// Mitsubishi GX Works2 project: PLCֹֹֹ_GROUP_31.docx   PLC: FX3G

// global labels: Global1
VAR_GLOBAL
  SW_DAY_START AT X007 : BOOL;
  RESET_ALL AT M10 : BOOL;
  DAY_ACTIVE AT M0 : BOOL;
  SW_EMERGENCY AT X005 : BOOL;
  LAMP_WORK_DAY AT Y007 : BOOL;
  INIT_RASPBERRY AT D1100 : REAL;
  INIT_LEMON AT D1110 : REAL;
  INIT_STABILIZER AT D1120 : REAL;
  INIT_GUMMIES AT D1130 : REAL;
  STOCK_RASPBERRY AT D1200 : REAL;
  STOCK_LEMON AT D1210 : REAL;
  STOCK_STABILIZER AT D1220 : REAL;
  STOCK_GUMMIES AT D1230 : REAL;
  SW_START_PROCESS AT X001 : BOOL;
  PHASE_PREPARE AT M2 : BOOL;
  PHASE_COOL AT M3 : BOOL;
  PHASE_MIX AT M4 : BOOL;
  ANALOG_IN1 AT D8280 : INT;
END_VAR
VAR_GLOBAL CONSTANT
  Constant_5 : REAL := 5;
END_VAR
VAR_GLOBAL
  TYPE_REGULAR AT M1 : BOOL;
END_VAR
VAR_GLOBAL CONSTANT
  Constant_6 : REAL := 6;
END_VAR
VAR_GLOBAL
  PROCESS_TRIGGER AT M6 : BOOL;
END_VAR
VAR_GLOBAL CONSTANT
  Constant_280 : REAL := 280;
  Constant_455 : REAL := 455;
  Constant_105 : REAL := 105;
  Constant_28 : REAL := 28;
  Constant_385 : REAL := 385;
  Constant_665 : REAL := 665;
  Constant_210 : REAL := 210;
  Constant_70 : REAL := 70;
END_VAR
VAR_GLOBAL
  NEEDED_RASPBERRY AT D1400 : REAL;
  NEEDED_LEMON AT D1410 : REAL;
  NEEDED_STABILIZER AT D1420 : REAL;
  NEEDED_GUMMIES AT D1430 : REAL;
  STOCK_OK AT M5 : BOOL;
  LAMP_PREPARE AT Y000 : BOOL;
  TIMER_PREPARE AT TC0 : BOOL;
  Const_5_sec AT K50 : INT;
  SW_COOL AT X002 : BOOL;
  PREP_RASPBERRY AT D1500 : REAL;
  PREP_LEMON AT D1510 : REAL;
  PREP_STABILIZER AT D1520 : REAL;
  PREP_GUMMIES AT D1530 : REAL;
END_VAR
VAR_GLOBAL CONSTANT
  Constant_35 : REAL := 35;
  Constant_420 : REAL := 420;
END_VAR
VAR_GLOBAL
  NEEDED_RASP_FOR_RASP AT D1800 : REAL;
  NEEDED_LEMON_FOR_RASP AT D1810 : REAL;
  NEEDED_STAB_FOR_RASP AT D1820 : REAL;
  NEEDED_LEMON_FOR_LEMON AT D1900 : REAL;
  NEEDED_STAB_FOR_LEMON AT D1910 : REAL;
END_VAR
VAR_GLOBAL CONSTANT
  Constant_560 : REAL := 560;
  Constant_140 : REAL := 140;
END_VAR
VAR_GLOBAL
  GELATO_RASPBERRY AT D1500 : REAL;
  GELATO_LEMON AT D1510 : REAL;
  COOL_GELATO_RASPBERRY AT D1600 : REAL;
END_VAR
VAR_GLOBAL CONSTANT
  Constant_0 : REAL;
END_VAR
VAR_GLOBAL
  TIMER_COOL AT TC1 : BOOL;
  Const_8_sec AT K80 : INT;
  LAMP_COOL AT Y002 : BOOL;
  TEMP_SENSOR AT X003 : BOOL;
  MIX_TOTAL AT D1700 : REAL;
  FLASH_DIFFERENCES AT M7 : BOOL;
  TIMER_MIX_3 AT TC2 : BOOL;
  Const_3_sec AT K30 : INT;
  LAMP_MIX_A AT Y005 : BOOL;
  Const_05_sec AT K5 : INT;
  TIMER_MIX_05 AT TC2 : BOOL;
  TIMER_MIX_050 AT TC3 : BOOL;
  LAMP_MIX_B AT Y006 : BOOL;
  TIMER_MIX AT TC4 : BOOL;
  STORAGE_COUNT AT D1300 : REAL;
END_VAR
VAR_GLOBAL CONSTANT
  Constant_1 : REAL := 1;
  Constant_10 : REAL := 10;
END_VAR
VAR_GLOBAL
  COOL_GELATO_LEMON AT D1610 : REAL;
  MANUAL_STOP_REQ AT M20 : BOOL;
  STOCK_STOP_REQ AT M21 : BOOL;
  MIX_TIMER_EN AT M8 : BOOL;
  TIMER_MIX_REGULAR AT TC4 : BOOL;
  TIMER_MIX_PINUK AT TC5 : BOOL;
  TS_2 AT TS2 : BOOL;
  TS_3 AT TS3 : BOOL;
  TS_5 AT TS5 : BOOL;
  TS_4 AT TS4 : BOOL;
  TIMER_MIX_REGUL AT TC4 : BOOL;
  TIMER_MIX_05_REGULAR AT TC2 : BOOL;
  TIMER_MIX_050_REGULAR AT TC3 : BOOL;
  TIMER_MIX_05_SPECIAL AT TC6 : BOOL;
  TIMER_MIX_050_SPECIAL AT TC7 : BOOL;
  Const_1_sec AT K10 : INT;
  TIMER_MIX_05_2 AT TC2 : BOOL;
  TIMER_MIX_05_3 AT TC3 : BOOL;
  INPUT AT D2000 : REAL;
END_VAR
VAR_GLOBAL CONSTANT
  Constant_400 : REAL := 400;
  WORD_0 : DINT;
END_VAR
VAR_GLOBAL
  ANALOG_OUT AT D8282 : DINT;
  UPDATE AT M8 : BOOL;
  STORAGE_OUT AT D1310 : REAL;
END_VAR
VAR_GLOBAL CONSTANT
  Constant_10_WORD : DINT := 10;
  Constant_40 : REAL := 40;
  Constant_5_5 : REAL := 5.5;
END_VAR

// task Task_01 (event TRUE, interval 0, priority 31): POU_01

PROGRAM POU_01
(* structured ladder/FBD written out as ST: instructions are called as NAME(EN, inputs, outputs); _pN, _eN, _tN stand for wires *)
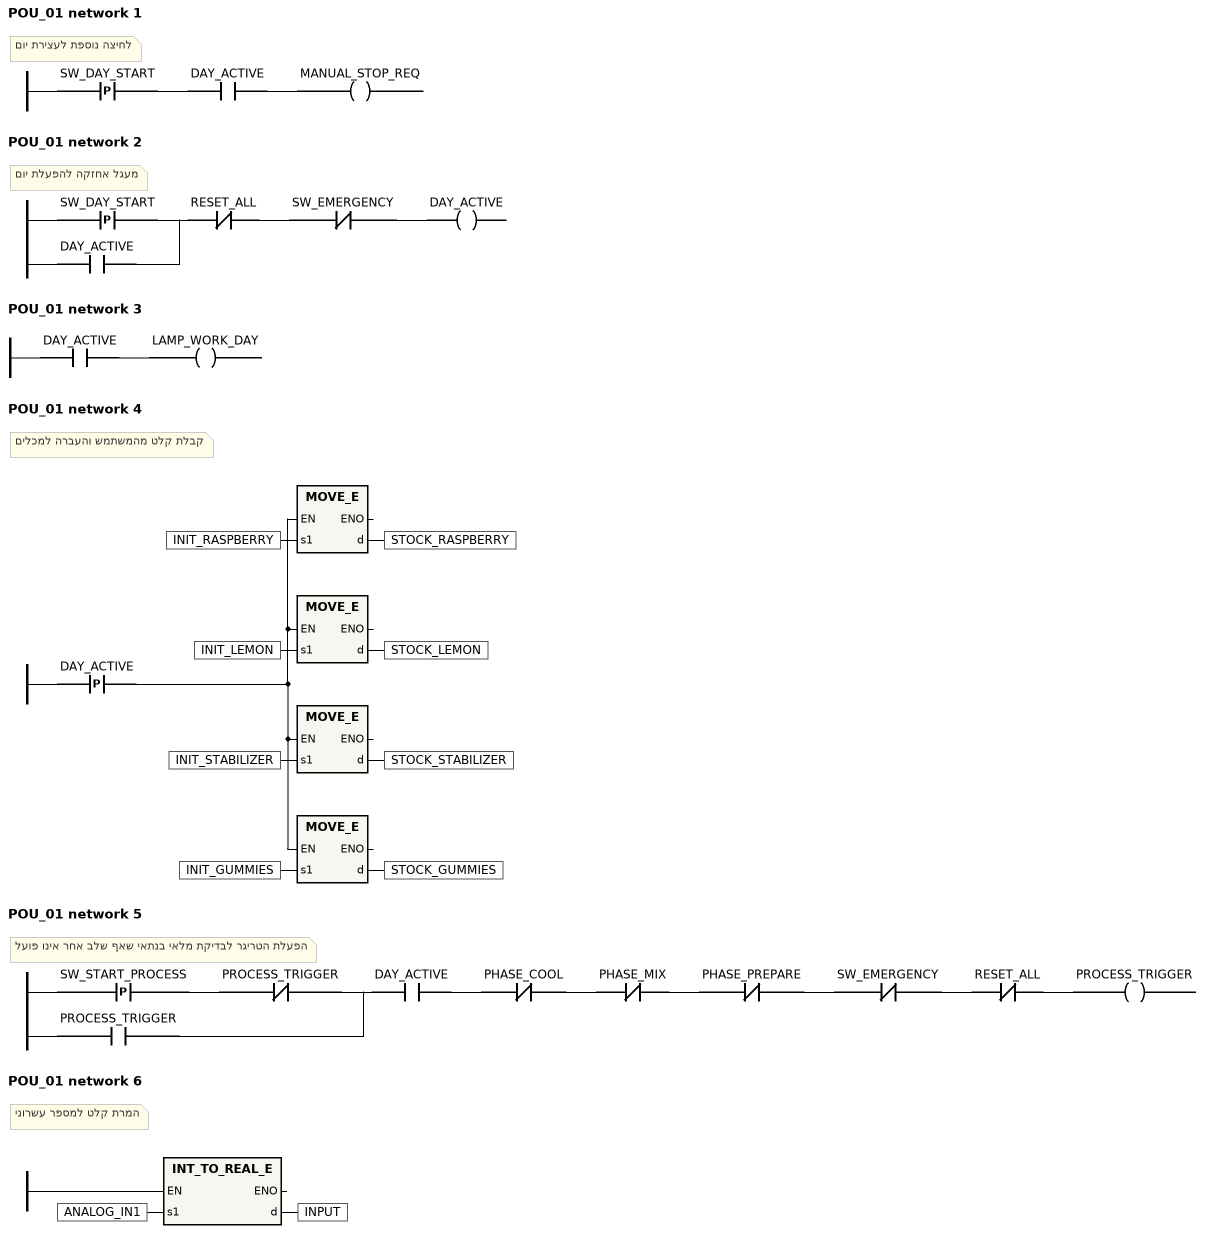
(* network 1 *)
(* לחיצה נוספת לעצירת יום *)
MANUAL_STOP_REQ := LDP(TRUE, SW_DAY_START) AND DAY_ACTIVE;
(* network 2 *)
(* מעגל אחזקה להפעלת יום *)
DAY_ACTIVE := ((LDP(TRUE, SW_DAY_START) OR DAY_ACTIVE) AND NOT RESET_ALL) AND NOT SW_EMERGENCY;
(* network 3 *)
LAMP_WORK_DAY := DAY_ACTIVE;
(* network 4 *)
(* קבלת קלט מהמשתמש והעברה למכלים *)
_p1 := LDP(TRUE, DAY_ACTIVE);
MOVE_E(_p1, INIT_RASPBERRY, STOCK_RASPBERRY);
MOVE_E(_p1, INIT_LEMON, STOCK_LEMON);
MOVE_E(_p1, INIT_STABILIZER, STOCK_STABILIZER);
MOVE_E(_p1, INIT_GUMMIES, STOCK_GUMMIES);
(* network 5 *)
(* הפעלת הטריגר לבדיקת מלאי בנתאי שאף שלב אחר אינו פועל *)
PROCESS_TRIGGER := (((((((LDP(TRUE, SW_START_PROCESS) AND NOT PROCESS_TRIGGER) OR PROCESS_TRIGGER) AND DAY_ACTIVE) AND NOT PHASE_COOL) AND NOT PHASE_MIX) AND NOT PHASE_PREPARE) AND NOT SW_EMERGENCY) AND NOT RESET_ALL;
(* network 6 *)
(* המרת קלט למספר עשרוני *)
INT_TO_REAL_E(TRUE, ANALOG_IN1, INPUT);
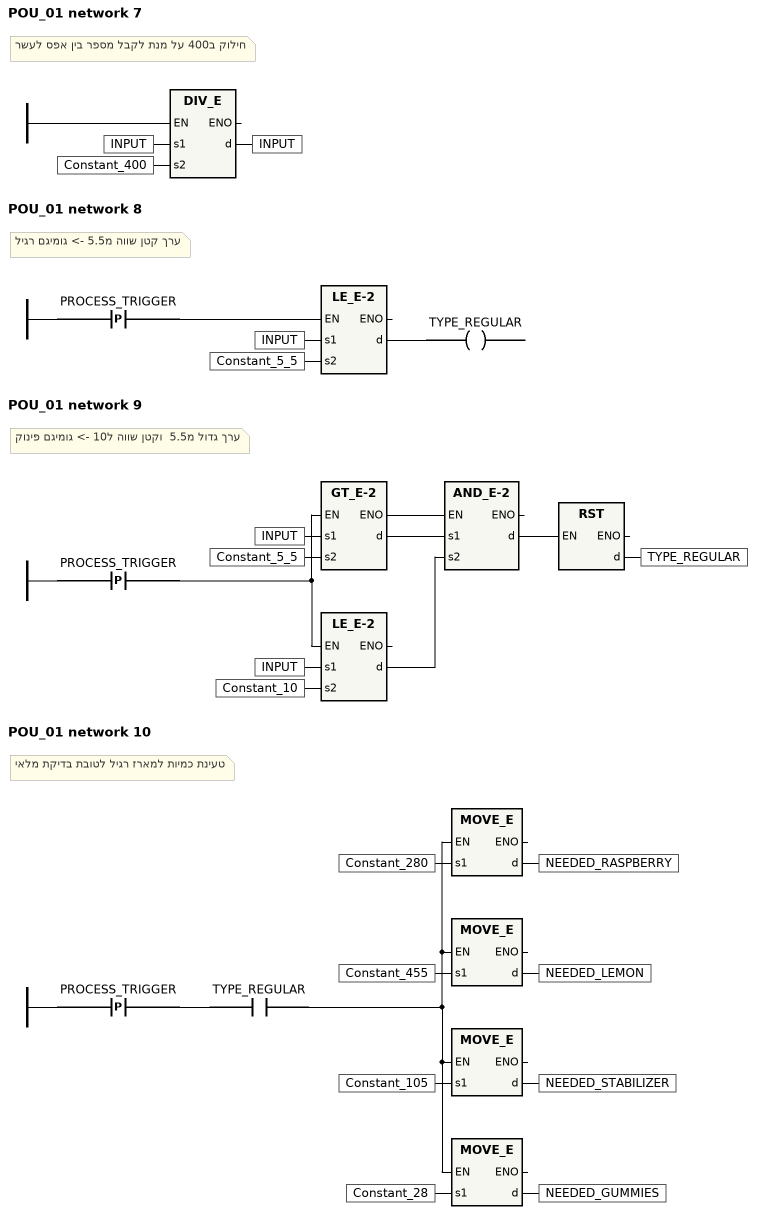
(* network 7 *)
(* חילוק ב400 על מנת לקבל מספר בין אפס לעשר *)
DIV_E(TRUE, INPUT, Constant_400, INPUT);
(* network 8 *)
(* ערך קטן שווה מ5.5 -> גומיגם רגיל *)
LE_E(LDP(TRUE, PROCESS_TRIGGER), INPUT, Constant_5_5, _t1);
TYPE_REGULAR := _t1;
(* network 9 *)
(* ערך גדול מ5.5  וקטן שווה ל10 -> גומיגם פינוק *)
_p1 := LDP(TRUE, PROCESS_TRIGGER);
_e3 := GT_E(_p1, INPUT, Constant_5_5, _t2);
LE_E(_p1, INPUT, Constant_10, _t4);
AND_E(_e3, _t2, _t4, _t5);
RST(_t5, TYPE_REGULAR);
(* network 10 *)
(* טעינת כמיות למארז רגיל לטובת בדיקת מלאי *)
_p1 := LDP(TRUE, PROCESS_TRIGGER) AND TYPE_REGULAR;
MOVE_E(_p1, Constant_280, NEEDED_RASPBERRY);
MOVE_E(_p1, Constant_455, NEEDED_LEMON);
MOVE_E(_p1, Constant_105, NEEDED_STABILIZER);
MOVE_E(_p1, Constant_28, NEEDED_GUMMIES);
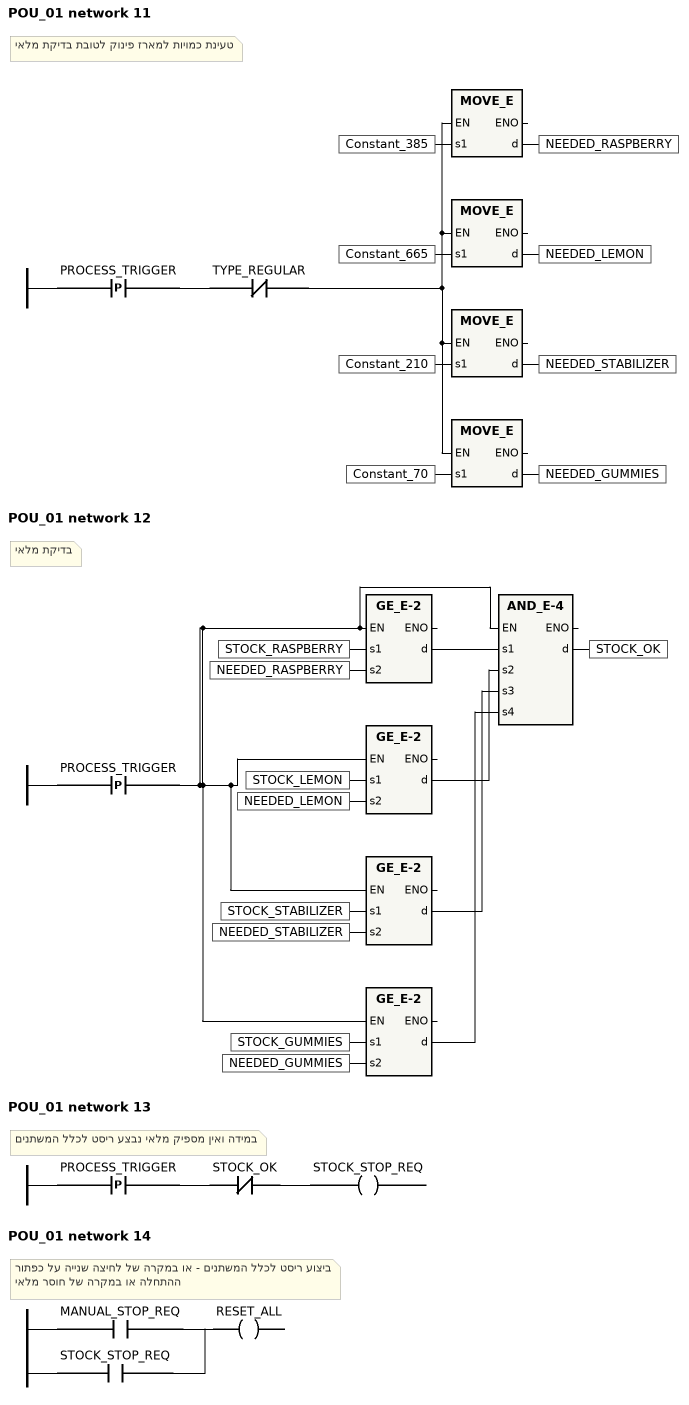
(* network 11 *)
(* טעינת כמויות למארז פינוק לטובת בדיקת מלאי *)
_p1 := LDP(TRUE, PROCESS_TRIGGER) AND NOT TYPE_REGULAR;
MOVE_E(_p1, Constant_385, NEEDED_RASPBERRY);
MOVE_E(_p1, Constant_665, NEEDED_LEMON);
MOVE_E(_p1, Constant_210, NEEDED_STABILIZER);
MOVE_E(_p1, Constant_70, NEEDED_GUMMIES);
(* network 12 *)
(* בדיקת מלאי *)
_p1 := LDP(TRUE, PROCESS_TRIGGER);
GE_E(_p1, STOCK_RASPBERRY, NEEDED_RASPBERRY, _t2);
GE_E(_p1, STOCK_LEMON, NEEDED_LEMON, _t3);
GE_E(_p1, STOCK_STABILIZER, NEEDED_STABILIZER, _t4);
GE_E(_p1, STOCK_GUMMIES, NEEDED_GUMMIES, _t5);
AND_E(_p1, _t2, _t3, _t4, _t5, STOCK_OK);
(* network 13 *)
(* במידה ואין מספיק מלאי נבצע ריסט לכלל המשתנים *)
STOCK_STOP_REQ := LDP(TRUE, PROCESS_TRIGGER) AND NOT STOCK_OK;
(* network 14 *)
(* ביצוע ריסט לכלל המשתנים - או במקרה של לחיצה שנייה על כפתור ההתחלה או במקרה של חוסר מלאי *)
RESET_ALL := MANUAL_STOP_REQ OR STOCK_STOP_REQ;
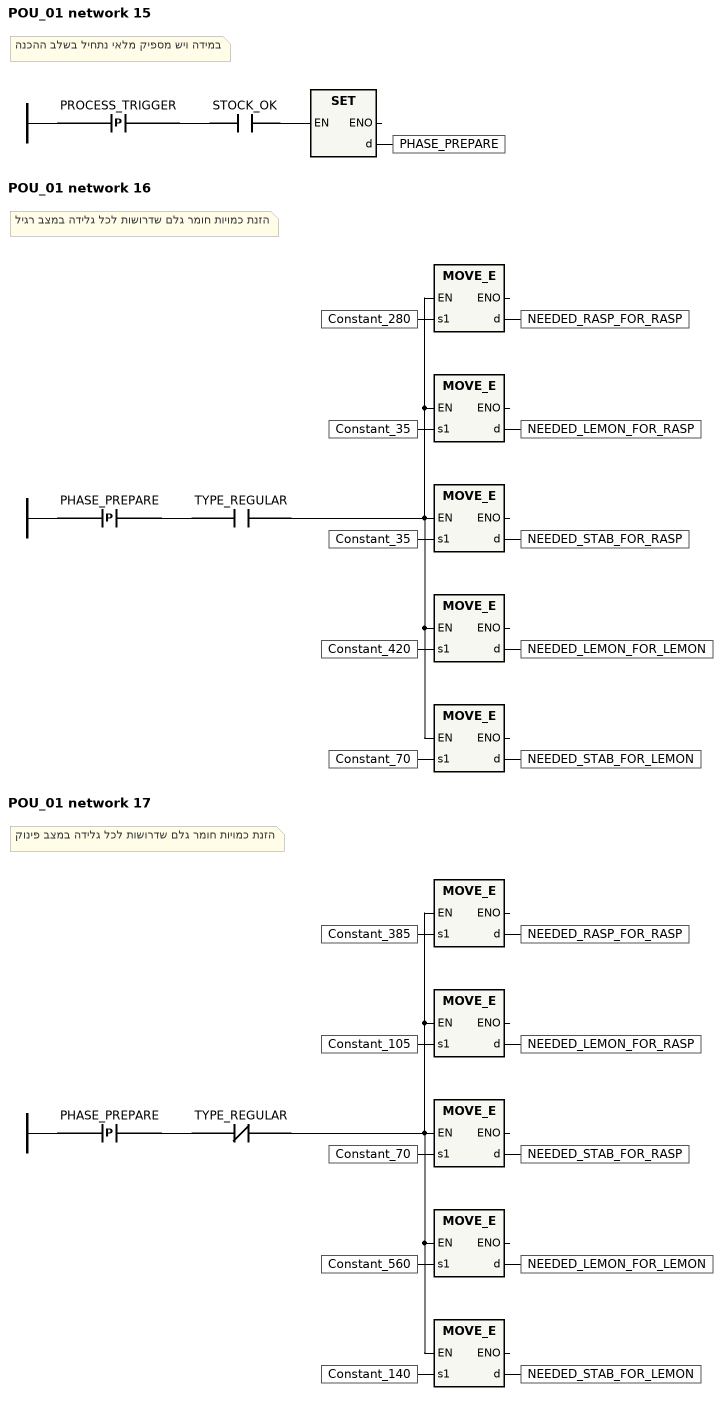
(* network 15 *)
(* במידה ויש מספיק מלאי נתחיל בשלב ההכנה *)
SET(LDP(TRUE, PROCESS_TRIGGER) AND STOCK_OK, PHASE_PREPARE);
(* network 16 *)
(* הזנת כמויות חומר גלם שדרושות לכל גלידה במצב רגיל *)
_p1 := LDP(TRUE, PHASE_PREPARE) AND TYPE_REGULAR;
MOVE_E(_p1, Constant_280, NEEDED_RASP_FOR_RASP);
MOVE_E(_p1, Constant_35, NEEDED_LEMON_FOR_RASP);
MOVE_E(_p1, Constant_35, NEEDED_STAB_FOR_RASP);
MOVE_E(_p1, Constant_420, NEEDED_LEMON_FOR_LEMON);
MOVE_E(_p1, Constant_70, NEEDED_STAB_FOR_LEMON);
(* network 17 *)
(* הזנת כמויות חומר גלם שדרושות לכל גלידה במצב פינוק *)
_p1 := LDP(TRUE, PHASE_PREPARE) AND NOT TYPE_REGULAR;
MOVE_E(_p1, Constant_385, NEEDED_RASP_FOR_RASP);
MOVE_E(_p1, Constant_105, NEEDED_LEMON_FOR_RASP);
MOVE_E(_p1, Constant_70, NEEDED_STAB_FOR_RASP);
MOVE_E(_p1, Constant_560, NEEDED_LEMON_FOR_LEMON);
MOVE_E(_p1, Constant_140, NEEDED_STAB_FOR_LEMON);
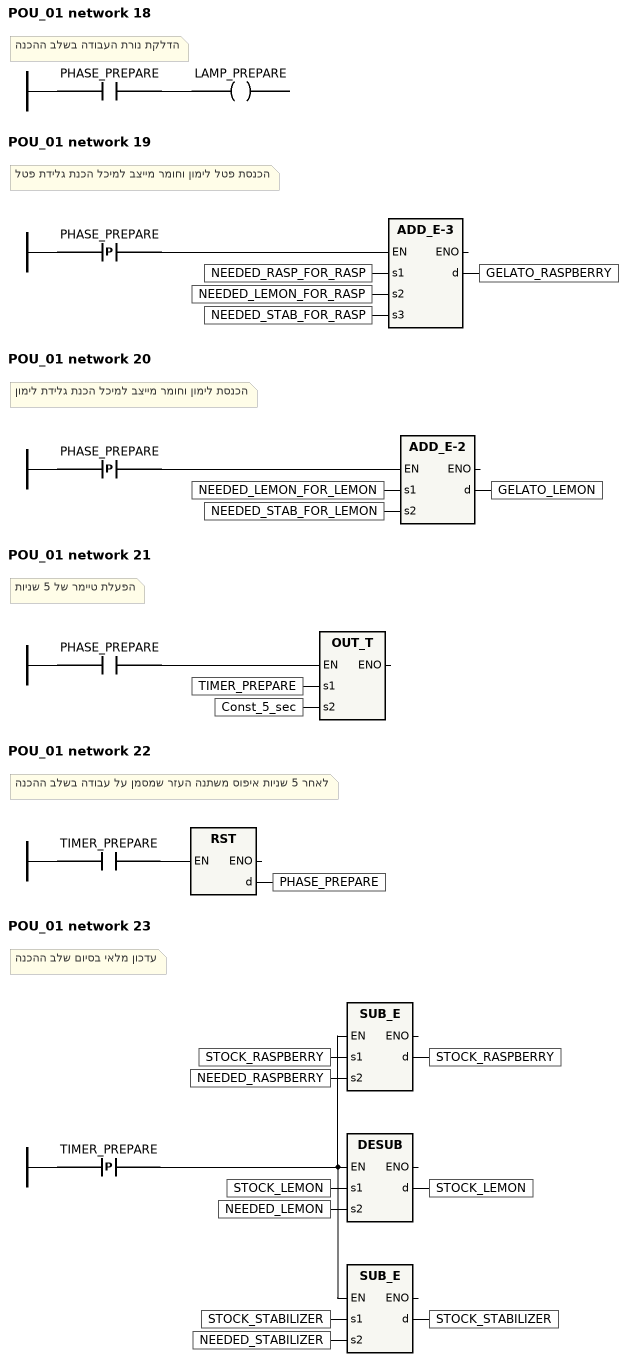
(* network 18 *)
(* הדלקת נורת העבודה בשלב ההכנה *)
LAMP_PREPARE := PHASE_PREPARE;
(* network 19 *)
(* הכנסת פטל לימון וחומר מייצב למיכל הכנת גלידת פטל *)
ADD_E(LDP(TRUE, PHASE_PREPARE), NEEDED_RASP_FOR_RASP, NEEDED_LEMON_FOR_RASP, NEEDED_STAB_FOR_RASP, GELATO_RASPBERRY);
(* network 20 *)
(* הכנסת לימון וחומר מייצב למיכל הכנת גלידת לימון *)
ADD_E(LDP(TRUE, PHASE_PREPARE), NEEDED_LEMON_FOR_LEMON, NEEDED_STAB_FOR_LEMON, GELATO_LEMON);
(* network 21 *)
(* הפעלת טיימר של 5 שניות *)
OUT_T(PHASE_PREPARE, TIMER_PREPARE, Const_5_sec);
(* network 22 *)
(* לאחר 5 שניות איפוס משתנה העזר שמסמן על עבודה בשלב ההכנה *)
RST(TIMER_PREPARE, PHASE_PREPARE);
(* network 23 *)
(* עדכון מלאי בסיום שלב ההכנה *)
_p1 := LDP(TRUE, TIMER_PREPARE);
SUB_E(_p1, STOCK_RASPBERRY, NEEDED_RASPBERRY, STOCK_RASPBERRY);
DESUB(_p1, STOCK_LEMON, NEEDED_LEMON, STOCK_LEMON);
SUB_E(_p1, STOCK_STABILIZER, NEEDED_STABILIZER, STOCK_STABILIZER);
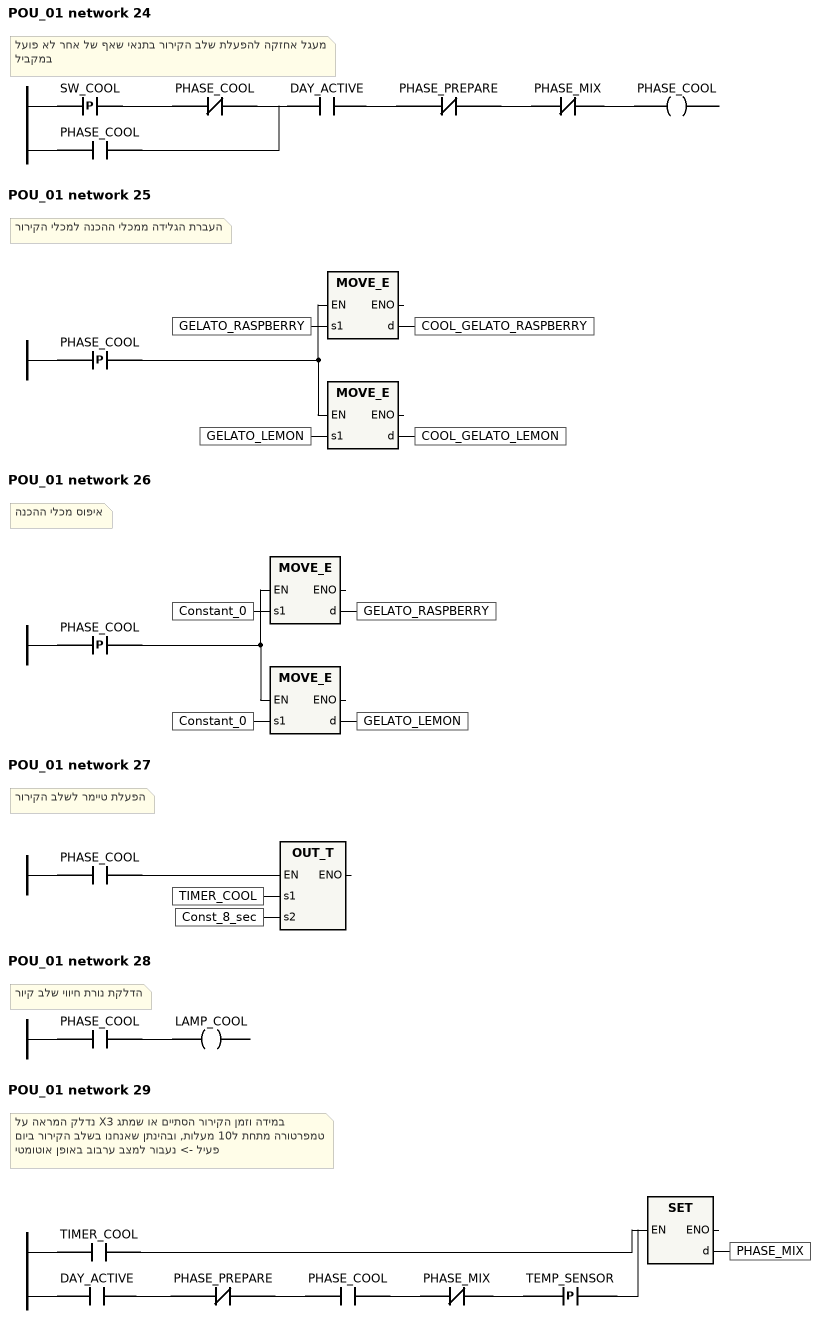
(* network 24 *)
(* מעגל אחזקה להפעלת שלב הקירור בתנאי שאף של אחר לא פועל במקביל *)
PHASE_COOL := ((((LDP(TRUE, SW_COOL) AND NOT PHASE_COOL) OR PHASE_COOL) AND DAY_ACTIVE) AND NOT PHASE_PREPARE) AND NOT PHASE_MIX;
(* network 25 *)
(* העברת הגלידה ממכלי ההכנה למכלי הקירור *)
_p1 := LDP(TRUE, PHASE_COOL);
MOVE_E(_p1, GELATO_RASPBERRY, COOL_GELATO_RASPBERRY);
MOVE_E(_p1, GELATO_LEMON, COOL_GELATO_LEMON);
(* network 26 *)
(* איפוס מכלי ההכנה *)
_p1 := LDP(TRUE, PHASE_COOL);
MOVE_E(_p1, Constant_0, GELATO_RASPBERRY);
MOVE_E(_p1, Constant_0, GELATO_LEMON);
(* network 27 *)
(* הפעלת טיימר לשלב הקירור *)
OUT_T(PHASE_COOL, TIMER_COOL, Const_8_sec);
(* network 28 *)
(* הדלקת נורת חיווי שלב קיור *)
LAMP_COOL := PHASE_COOL;
(* network 29 *)
(* במידה וזמן הקירור הסתיים או שמתג X3 נדלק המראה על טמפרטורה מתחת ל10 מעלות, ובהינתן שאנחנו בשלב הקירור ביום פעיל -> נעבור למצב ערבוב באופן אוטומטי *)
SET(TIMER_COOL OR (DAY_ACTIVE AND NOT PHASE_PREPARE AND PHASE_COOL AND NOT PHASE_MIX AND LDP(TRUE, TEMP_SENSOR)), PHASE_MIX);
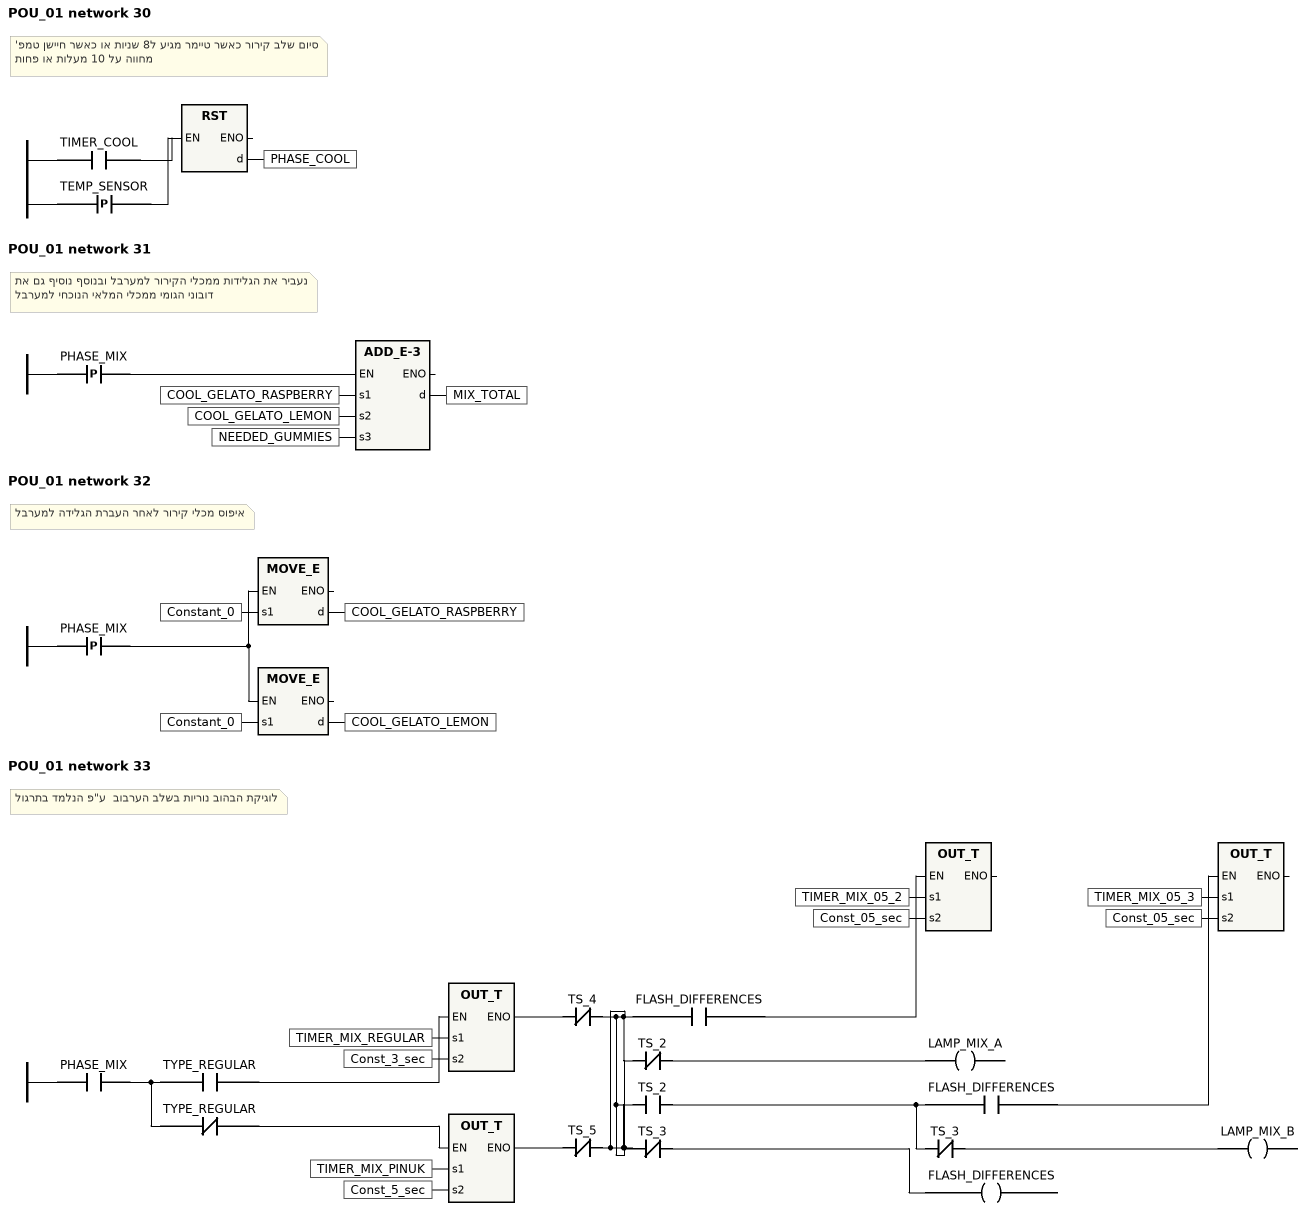
(* network 30 *)
(* סיום שלב קירור כאשר טיימר מגיע ל8 שניות או כאשר חיישן טמפ' מחווה על 10 מעלות או פחות *)
RST(TIMER_COOL OR LDP(TRUE, TEMP_SENSOR), PHASE_COOL);
(* network 31 *)
(* נעביר את הגלידות ממכלי הקירור למערבל ובנוסף נוסיף גם את דובוני הגומי ממכלי המלאי הנוכחי למערבל *)
ADD_E(LDP(TRUE, PHASE_MIX), COOL_GELATO_RASPBERRY, COOL_GELATO_LEMON, NEEDED_GUMMIES, MIX_TOTAL);
(* network 32 *)
(* איפוס מכלי קירור לאחר העברת הגלידה למערבל *)
_p1 := LDP(TRUE, PHASE_MIX);
MOVE_E(_p1, Constant_0, COOL_GELATO_RASPBERRY);
MOVE_E(_p1, Constant_0, COOL_GELATO_LEMON);
(* network 33 *)
(* לוגיקת הבהוב נוריות בשלב הערבוב  ע"פ הנלמד בתרגול *)
_e1 := OUT_T(PHASE_MIX AND TYPE_REGULAR, TIMER_MIX_REGULAR, Const_3_sec);
_e2 := OUT_T(PHASE_MIX AND NOT TYPE_REGULAR, TIMER_MIX_PINUK, Const_5_sec);
_p3 := (_e1 AND NOT TS_4) OR (_e2 AND NOT TS_5);
OUT_T(_p3 AND FLASH_DIFFERENCES, TIMER_MIX_05_2, Const_05_sec);
LAMP_MIX_A := _p3 AND NOT TS_2;
_p4 := _p3 AND TS_2;
OUT_T(_p4 AND FLASH_DIFFERENCES, TIMER_MIX_05_3, Const_05_sec);
LAMP_MIX_B := _p4 AND NOT TS_3;
FLASH_DIFFERENCES := _p3 AND NOT TS_3;
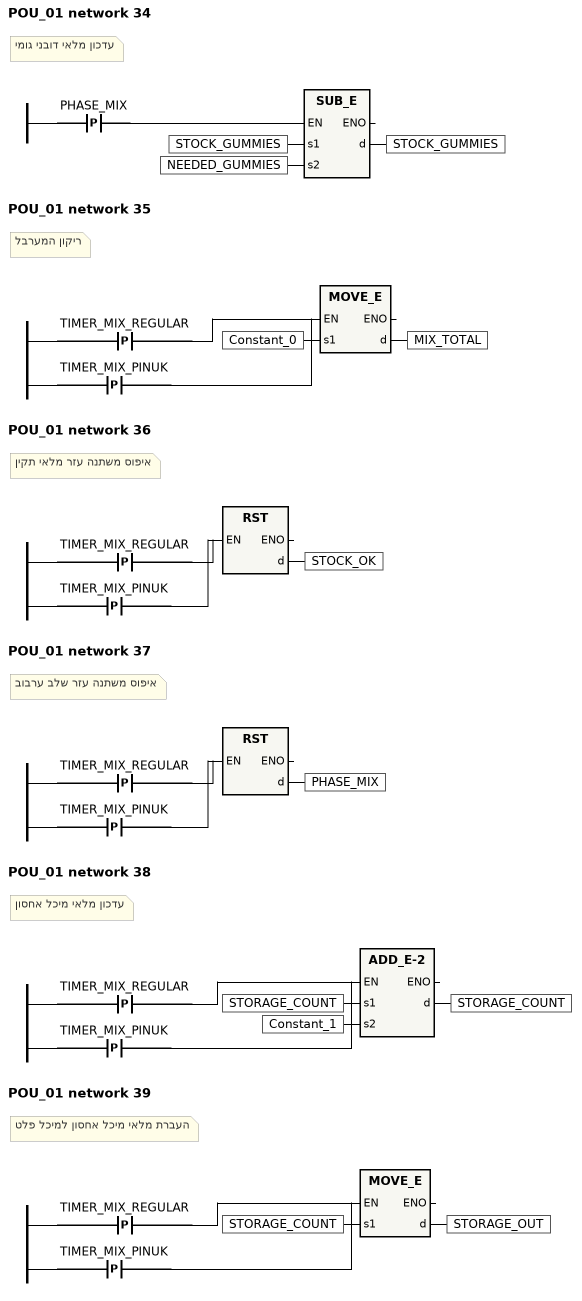
(* network 34 *)
(* עדכון מלאי דובני גומי *)
SUB_E(LDP(TRUE, PHASE_MIX), STOCK_GUMMIES, NEEDED_GUMMIES, STOCK_GUMMIES);
(* network 35 *)
(* ריקון המערבל *)
MOVE_E(LDP(TRUE, TIMER_MIX_REGULAR) OR LDP(TRUE, TIMER_MIX_PINUK), Constant_0, MIX_TOTAL);
(* network 36 *)
(* איפוס משתנה עזר מלאי תקין *)
RST(LDP(TRUE, TIMER_MIX_REGULAR) OR LDP(TRUE, TIMER_MIX_PINUK), STOCK_OK);
(* network 37 *)
(* איפוס משתנה עזר שלב ערבוב *)
RST(LDP(TRUE, TIMER_MIX_REGULAR) OR LDP(TRUE, TIMER_MIX_PINUK), PHASE_MIX);
(* network 38 *)
(* עדכון מלאי מיכל אחסון *)
ADD_E(LDP(TRUE, TIMER_MIX_REGULAR) OR LDP(TRUE, TIMER_MIX_PINUK), STORAGE_COUNT, Constant_1, STORAGE_COUNT);
(* network 39 *)
(* העברת מלאי מיכל אחסון למיכל פלט *)
MOVE_E(LDP(TRUE, TIMER_MIX_REGULAR) OR LDP(TRUE, TIMER_MIX_PINUK), STORAGE_COUNT, STORAGE_OUT);
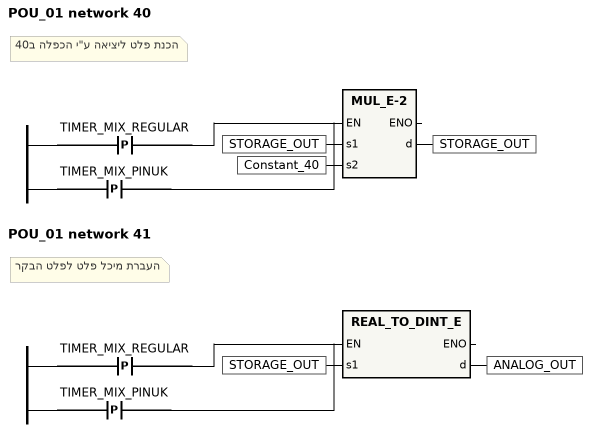
(* network 40 *)
(* הכנת פלט ליציאה ע"י הכפלה ב40 *)
MUL_E(LDP(TRUE, TIMER_MIX_REGULAR) OR LDP(TRUE, TIMER_MIX_PINUK), STORAGE_OUT, Constant_40, STORAGE_OUT);
(* network 41 *)
(* העברת מיכל פלט לפלט הבקר *)
REAL_TO_DINT_E(LDP(TRUE, TIMER_MIX_REGULAR) OR LDP(TRUE, TIMER_MIX_PINUK), STORAGE_OUT, ANALOG_OUT);
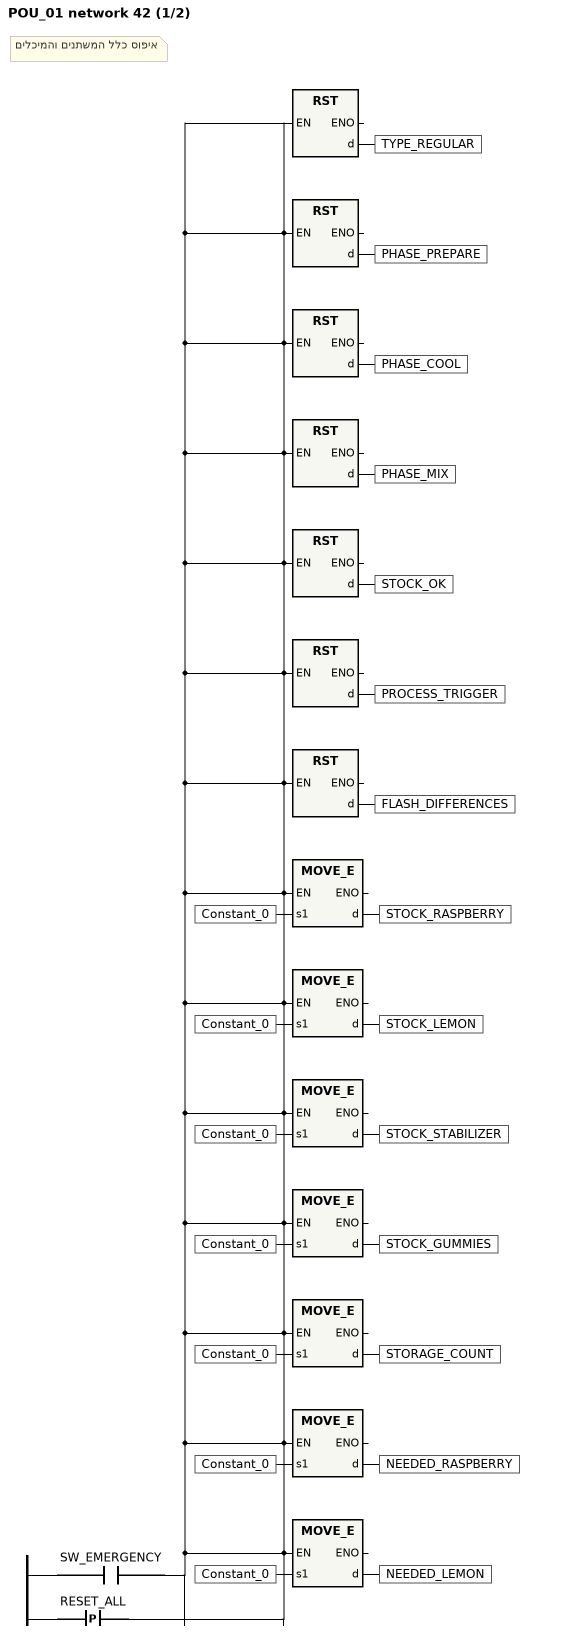
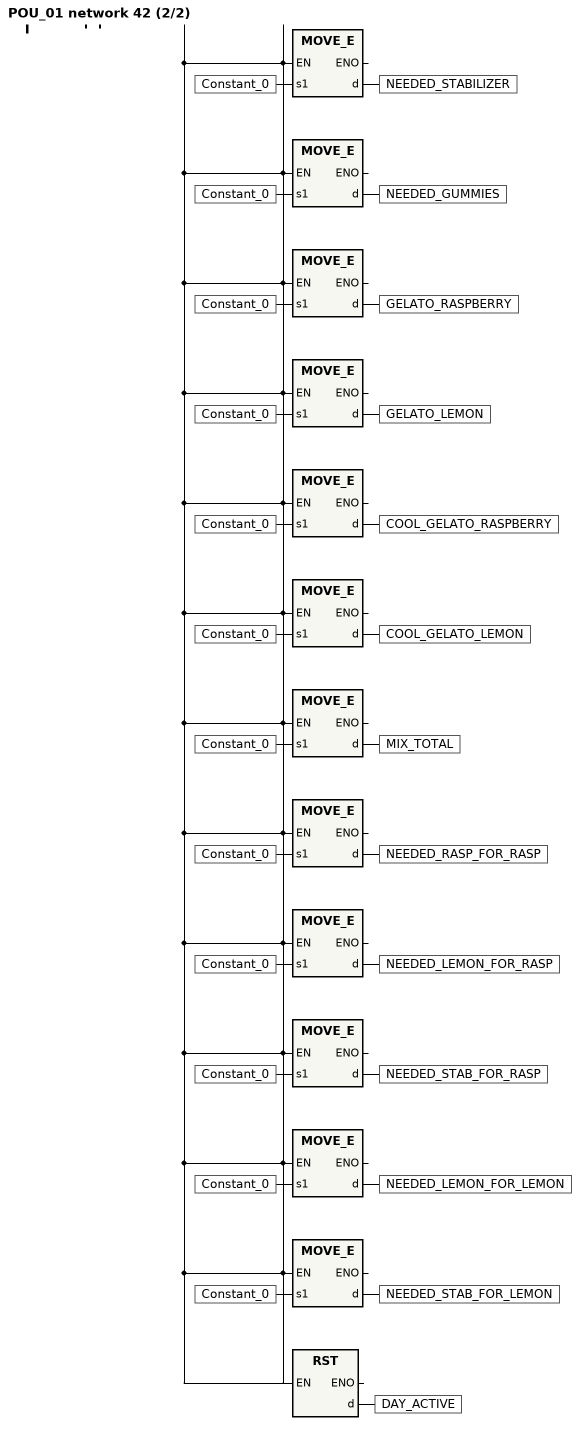
(* network 42 *)
(* איפוס כלל המשתנים והמיכלים *)
_p1 := SW_EMERGENCY OR LDP(TRUE, RESET_ALL);
RST(_p1, TYPE_REGULAR);
RST(_p1, PHASE_PREPARE);
RST(_p1, PHASE_COOL);
RST(_p1, PHASE_MIX);
RST(_p1, STOCK_OK);
RST(_p1, PROCESS_TRIGGER);
RST(_p1, FLASH_DIFFERENCES);
MOVE_E(_p1, Constant_0, STOCK_RASPBERRY);
MOVE_E(_p1, Constant_0, STOCK_LEMON);
MOVE_E(_p1, Constant_0, STOCK_STABILIZER);
MOVE_E(_p1, Constant_0, STOCK_GUMMIES);
MOVE_E(_p1, Constant_0, STORAGE_COUNT);
MOVE_E(_p1, Constant_0, NEEDED_RASPBERRY);
MOVE_E(_p1, Constant_0, NEEDED_LEMON);
MOVE_E(_p1, Constant_0, NEEDED_STABILIZER);
MOVE_E(_p1, Constant_0, NEEDED_GUMMIES);
MOVE_E(_p1, Constant_0, GELATO_RASPBERRY);
MOVE_E(_p1, Constant_0, GELATO_LEMON);
MOVE_E(_p1, Constant_0, COOL_GELATO_RASPBERRY);
MOVE_E(_p1, Constant_0, COOL_GELATO_LEMON);
MOVE_E(_p1, Constant_0, MIX_TOTAL);
MOVE_E(_p1, Constant_0, NEEDED_RASP_FOR_RASP);
MOVE_E(_p1, Constant_0, NEEDED_LEMON_FOR_RASP);
MOVE_E(_p1, Constant_0, NEEDED_STAB_FOR_RASP);
MOVE_E(_p1, Constant_0, NEEDED_LEMON_FOR_LEMON);
MOVE_E(_p1, Constant_0, NEEDED_STAB_FOR_LEMON);
RST(_p1, DAY_ACTIVE);
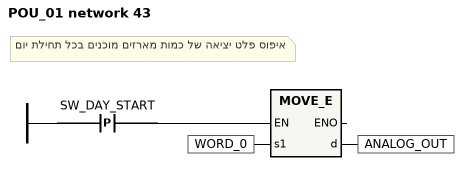
(* network 43 *)
(* איפוס פלט יציאה של כמות מארזים מוכנים בכל תחילת יום *)
MOVE_E(LDP(TRUE, SW_DAY_START), WORD_0, ANALOG_OUT);
END_PROGRAM
